FUNCTION_BLOCK FB_LamparaIntermitente_IL
// La lampara parpadea de forma continua
VAR_INPUT
    TiempoParpadeo: TIME := T#500MS;
END_VAR
VAR
    Temporizador: TON;
    Lampara AT %Q*: BOOL;
END_VAR

// NETWORK 1
// Temporizador auto-pilotado
// instruction list
CAL     Temporizador(
    IN      := NOT Temporizador.Q
    PT      := TiempoParpadeo)

// NETWORK 2
// instruction list
LD      Temporizador.Q
JMPCN   End

// NETWORK 3
// Salida conmutada
// instruction list
LD      Lampara
STN     Lampara

// NETWORK 4
End:
// instruction list

END_FUNCTION_BLOCK

(* stored: Version 1.1.0.1, ProductVersion 3.1.4024.15
   POU FB_LamparaIntermitente_IL: Id {ce178025-ba9a-4fc2-92f6-70b394b9bdde}, SpecialFunc None *)
